TYPE DUT_SKILL_INPUT :
STRUCT
	///Range of parameters
	ParameterInput: ARRAY[0..ParameterCnt] OF DUT_PARAMETER_INPUT;
	///Start process
	Execute: BOOL;
END_STRUCT
END_TYPE

(* stored: Version 1.1.0.1, ProductVersion 3.1.0.25
   DUT DUT_SKILL_INPUT: Id {e7429fba-517c-4317-a140-0bf8ff3d0c59} *)
